FUNCTION_BLOCK FB_teknicMotorEC
VAR
	//I/O
	bBrake			AT %Q*  : BOOL;
	bHomeSensor		AT %I*  : BOOL;
	bClampSensor 	AT %I*  : BOOL;
	fHeightDisp				: REAL;
	
	//Init
	bMotorInverted : BOOL;
	bMotorDisables : BOOL;
	
	fMoveAccl 		: LREAL := 50;
	fMoveDcl 		: LREAL := 50;
	fMoveVelocity 	: LREAL;
	
	torqueVelocity		: LREAL;
	torqueAcceleration	: LREAL;
	torqueDeceleration	: LREAL;
	
	homeVelocity		: LREAL;
	homeSetPosition		: LREAL;
	homeTorqueLimit		: LREAL;
	
	jogTorque			: LREAL;
	
	//State Var
	nMoveState 				: INT;
	nMoveStateTorque		: INT;
	nHomeState				: INT;
	nInitState 				: INT;
	nResetState 			: INT;
	estopState 				: INT := 0; // 0 = Idle, 3 = GearOut, 2 = Stop, 1 = Done
	stopState				: INT;
	
	bIdle 					: BOOL;
	bIdleEnabled 			: BOOL;
	bIdleDisabled 			: BOOL;
	
	fMinHeight				: REAL;
	fMaxHeight 				: REAL := 115;
	fPrevHeight				: REAL;
	bSensorWarning			: BOOL;
	fHeight					: REAL;
	nMoveUpCount			: INT;
	nMoveDownCount			: INT;

	stError : ST_errorRef;
	
	// Timer to turn brake on if motor is left holding carriage for so long;
	fbBrakeTimer 	: TON;
	bIn				: BOOL;
	tPt				: TIME := T#1M;
	bQ				: BOOL;
	tEt				: TIME;
	
	/////////// EC Motor //////////////////////////////////
	fbMotor : axis_REF;
	
	//Power
	fbMotorPower	: MC_Power;
	stMotorPowerOut : ST_McOutputs;
	
	//Reset
	fbMotorReset 	: MC_RESET;
	stMotorResetOut : ST_McOutputs;

	//Halt
	fbMotorHalt 	: MC_HALT;
	stMotorHaltOut 	: ST_McOutputs;
	
	//Velocity Jog
	fbMotorJog 		: MC_JOG;
	stMotorJogOut 	: ST_McOutputs;
	eJogMode 		: E_JogMode;
	nJogModeSelect 	: INT := 2;
	

	//Homing
	fbMotorHome		: MC_Home;
	stHomingOptions : ST_HomingOptions;
	stMotorHomeOut 	: ST_McOutputs;
	bDummyHomingCam : BOOL;
	stHomingMode 	: MC_HomingMode;
	bCheckhomeSensor: BOOL;
	bMotorHomeStatus: BOOL;
	bHomeSensorTriggered : BOOL;
	fbFreeSensorTimer : TON;
	
	//Mode
	fbMotorWriteMode	: MC_WriteDriveOperationMode;
	stMotorWriteModeOut : ST_McOutputs;
	fbMotorReadMode		: MC_ReadDriveOperationMode;
	stMotorReadModeOut 	: ST_McOutputs;
	stOpModeMotor 		: E_DriveOperationMode;
	stOpModeMotorInt	: DINT;
	stWriteMode 		: E_DriveOperationMode;
	nWriteModeSelect 	: DINT := 0;
	fbReadBoolParam		: MC_readParameter;
	fbReadRealParam		: MC_readParameter;
	stReadParamOut 		: ST_mcOutputs;
	eParameter 			: MC_AxisParameter; //Parameter to read or write. https://infosys.beckhoff.com/english.php?content=../content/1033/tcplclib_tc2_mc2/70069259.html&id=
	fReadValue 			: LREAL; // Return value when MC_AxisParameter is of type REAL
	bReadValue 			: LREAL; // Return value when MC_AxisParameter is of type BOOL
	fbWriteRealParam	: MC_WriteParameter;
	fbWriteBoolParam	: MC_WriteParameter;
	stWriteParameterOut : ST_mcOutputs;
	fWriteValue 		: LREAL; // Write value when MC_AxisParameter is of type REAL
	bWriteValue			: BOOL; // Write value when MC_AxisParameter is of type BOOL
	
	//Move Absolute
	fbMotorMoveAbsolute		: MC_MoveAbsolute;
	stMotorMoveAbsoluteOut 	: ST_mcOutputs;
	bChangePosition 		: BOOL;
	fPosition 				: LREAL := 300;
	fStartPos				: LREAL;
	fHalfwayPos				: LREAL;
	
	//Move Relative
	fbMotorMoveRelative		: MC_MoveRelative;
	stMotorMoveRelativeOut 	: ST_McOutputs;
	
	//Move Velocity
	fbMotorMoveVelocity		: MC_MoveVelocity;
	stMotorMoveVelocityOut	: ST_mcOutputs;
	fVel 					: LREAL := 100;
	stDirection 			: MC_Direction;
	stDirectionSelect 		: INT := 1;

	// Stop
	fbMotorStop		: MC_Stop;
	stMotorStopOut 	: ST_mcOutputs;
	bExectuteStop 	: BOOL;
	bStopDone 		: BOOL;
	bStopBtn 		: BOOL;
	
	//Torque
	fbMotorTorque		: FB_moveToTorque;
	stMotorTorqueOut 	: ST_mcOutputs;
	fTorque 			: LREAL := 2;
	torqueDirection		: INT;
	torqueTime			: TIME := T#200MS;

	
	//Gear Coupling
	fbMotorGearIn : MC_GearIn;
	fbMotorGearOut: MC_GearOut;
	stMotorGearInOut : ST_McOutputs;
	stMotorGearOutOut: ST_McOutputs;
	refMasterAxis : axis_REF;
	
	//Status
	fbMotorReadStatus 		: MC_ReadStatus;
	stMotorStatus 			: ST_AxisStatus;
	stMotorReadStatusOut 	: ST_mcOutputs;
	
	//Set Position
	fbMotorSetPosition			: MC_SetPosition;
	stMotorSetPositionOut 		: ST_mcOutputs;
	stMotorSetPositionOption 	: ST_SetPositionOptions;

	fbMotorWriteParameter	: MC_WriteParameter;
	stMotorWriteOut 		: ST_mcOutputs;
	
	sModeDisp 		: STRING;
	fbReadModeTimer	: TON;
		
	fbHomeToTorque		: FB_homeToTorque;
	stHomeToTorqueOut 	: ST_mcOutputs;
	direction			: INT; // 0- PositiveDirection, 1- NegativeDirection
	homeTimeLimit		: TIME := T#2M;
	//homeBackOffPos		: LREAL := 1.5;
	homeBackOffPos		: LREAL := 10;

	bUsingStopReset: BOOL;
END_VAR

(* Behavior of this motor setup is a steady state of disabling the motor when no command is being executed. This setup is best with motors that have a brake
connected to the PLC or motors connected to systems where the system can remain still without assistance from the motor. 
*)
fbBrakeTimer(IN:= bIn, PT:= tPt, Q=> bQ, ET=> tEt);
IF GVL_machine.bMotorsInitialized AND nResetState = 0 THEN
	//bUsingStopReset := FALSE;
	IF bIdleDisabled THEN 
		bIn := TRUE;
	ELSE
		bIn := FALSE;
	END_IF
	
	IF bQ THEN
		IF fbMotor.status.HasJob THEN 
			bIn := FALSE;
		ELSE
			stop();
			brakeOn();
		END_IF
		
	END_IF
	
	(*IF bIdle THEN
		bIdleDisabled R= bIdle;
		bIdleEnabled S= SEL(stop() = 1,FALSE,TRUE);
	ELSE
		bIdleEnabled R= NOT bIdle;
		bIdleDisabled S= SEL(removeStop() = 1,FALSE,TRUE);
	END_IF*)
	IF bIdle THEN
		bIdleDisabled R= bIdle;
		IF (fbMotor.Status.HasBeenStopped OR fbMotor.Status.StandStill) AND bIdleEnabled THEN
			stopState := 0;
			fbMotorStop.Execute := FALSE;
		ELSE
			bIdleEnabled := SEL(stop() = 1,FALSE,TRUE);
			//bUsingStopReset := TRUE;
		END_IF
	ELSE
		bIdleEnabled R= NOT bIdle;
		IF (fbMotor.Status.HasBeenStopped OR fbMotor.Status.StandStill) AND NOT bIdleDisabled THEN
			bIdleDisabled := SEL(removeStop() = 1,FALSE,TRUE);
		ELSE
			stopState := 0;
		END_IF
	END_IF
END_IF

	
actPower();
actHome();
actMode();
actStop();
actMove();
actTorque();
actCouple();
actStatus();


fbMotor();
fbMotorJog.JogForward := FALSE;
fbMotorJog.JogBackwards := FALSE;

ACTION actCouple:
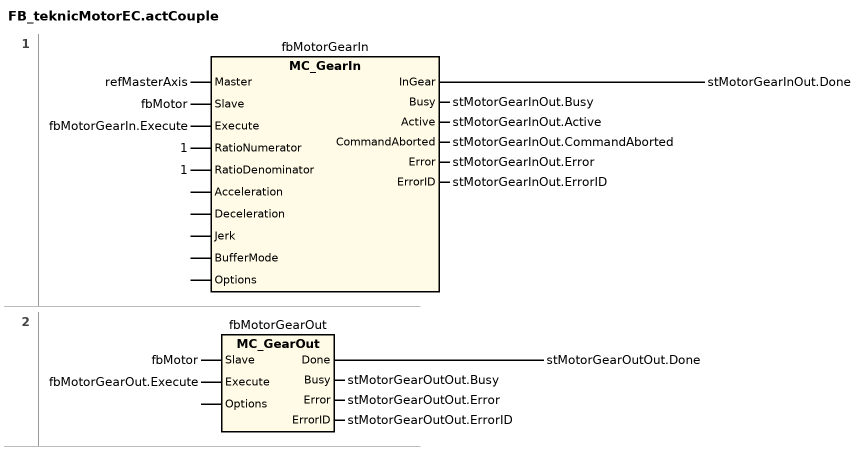
// NETWORK 1
fbMotorGearIn(
    Master := refMasterAxis,
    Slave := fbMotor,
    Execute := fbMotorGearIn.Execute,
    RatioNumerator := 1,
    RatioDenominator := 1,
    Busy => stMotorGearInOut.Busy,
    Active => stMotorGearInOut.Active,
    CommandAborted => stMotorGearInOut.CommandAborted,
    Error => stMotorGearInOut.Error,
    ErrorID => stMotorGearInOut.ErrorID); // MC_GearIn
stMotorGearInOut.Done := fbMotorGearIn.InGear;

// NETWORK 2
fbMotorGearOut(
    Slave := fbMotor,
    Execute := fbMotorGearOut.Execute,
    Busy => stMotorGearOutOut.Busy,
    Error => stMotorGearOutOut.Error,
    ErrorID => stMotorGearOutOut.ErrorID); // MC_GearOut
stMotorGearOutOut.Done := fbMotorGearOut.Done;
END_ACTION

ACTION actHome:
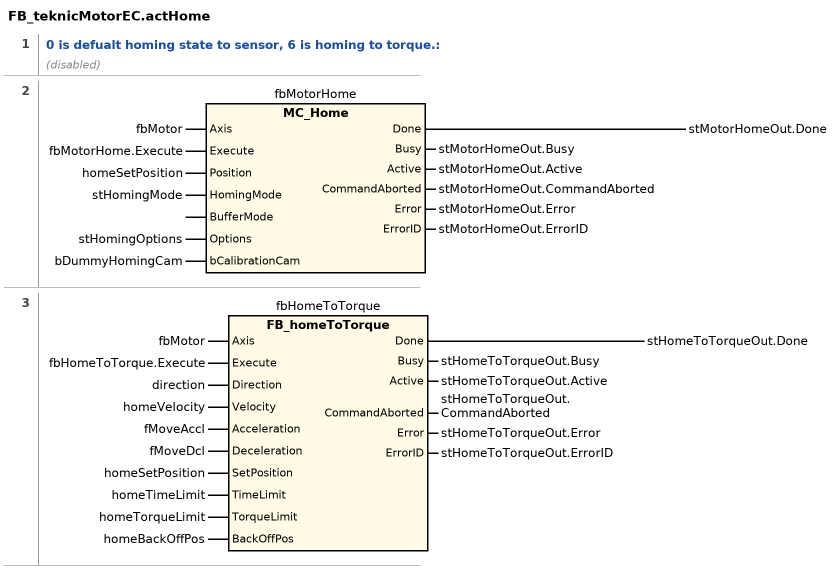
// NETWORK 1 (disabled)
// label: 0 is defualt homing state to sensor, 6 is homing to torque.

// NETWORK 2
fbMotorHome(
    Axis := fbMotor,
    Execute := fbMotorHome.Execute,
    Position := homeSetPosition,
    HomingMode := stHomingMode,
    Options := stHomingOptions,
    bCalibrationCam := bDummyHomingCam,
    Busy => stMotorHomeOut.Busy,
    Active => stMotorHomeOut.Active,
    CommandAborted => stMotorHomeOut.CommandAborted,
    Error => stMotorHomeOut.Error,
    ErrorID => stMotorHomeOut.ErrorID); // MC_Home
stMotorHomeOut.Done := fbMotorHome.Done;

// NETWORK 3
fbHomeToTorque(
    Axis := fbMotor,
    Execute := fbHomeToTorque.Execute,
    Direction := direction,
    Velocity := homeVelocity,
    Acceleration := fMoveAccl,
    Deceleration := fMoveDcl,
    SetPosition := homeSetPosition,
    TimeLimit := homeTimeLimit,
    TorqueLimit := homeTorqueLimit,
    BackOffPos := homeBackOffPos,
    Busy => stHomeToTorqueOut.Busy,
    Active => stHomeToTorqueOut.Active,
    CommandAborted => stHomeToTorqueOut.CommandAborted,
    Error => stHomeToTorqueOut.Error,
    ErrorID => stHomeToTorqueOut.ErrorID); // FB_homeToTorque
stHomeToTorqueOut.Done := fbHomeToTorque.Done;
END_ACTION

ACTION actMode:
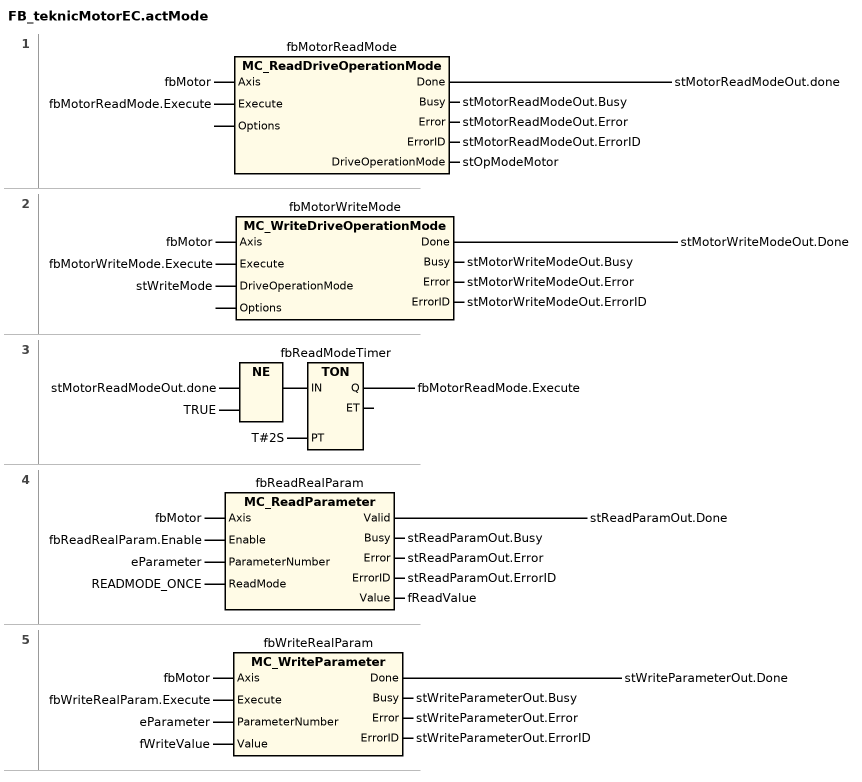
// NETWORK 1
fbMotorReadMode(
    Axis := fbMotor,
    Execute := fbMotorReadMode.Execute,
    Busy => stMotorReadModeOut.Busy,
    Error => stMotorReadModeOut.Error,
    ErrorID => stMotorReadModeOut.ErrorID,
    DriveOperationMode => stOpModeMotor); // MC_ReadDriveOperationMode
stMotorReadModeOut.done := fbMotorReadMode.Done;

// NETWORK 2
fbMotorWriteMode(
    Axis := fbMotor,
    Execute := fbMotorWriteMode.Execute,
    DriveOperationMode := stWriteMode,
    Busy => stMotorWriteModeOut.Busy,
    Error => stMotorWriteModeOut.Error,
    ErrorID => stMotorWriteModeOut.ErrorID); // MC_WriteDriveOperationMode
stMotorWriteModeOut.Done := fbMotorWriteMode.Done;

// NETWORK 3
fbReadModeTimer(IN := stMotorReadModeOut.done <> TRUE, PT := T#2S); // TON
fbMotorReadMode.Execute := fbReadModeTimer.Q;

// NETWORK 4
fbReadRealParam(
    Axis := fbMotor,
    Enable := fbReadRealParam.Enable,
    ParameterNumber := eParameter,
    ReadMode := READMODE_ONCE,
    Busy => stReadParamOut.Busy,
    Error => stReadParamOut.Error,
    ErrorID => stReadParamOut.ErrorID,
    Value => fReadValue); // MC_ReadParameter
stReadParamOut.Done := fbReadRealParam.Valid;

// NETWORK 5
fbWriteRealParam(
    Axis := fbMotor,
    Execute := fbWriteRealParam.Execute,
    ParameterNumber := eParameter,
    Value := fWriteValue,
    Busy => stWriteParameterOut.Busy,
    Error => stWriteParameterOut.Error,
    ErrorID => stWriteParameterOut.ErrorID); // MC_WriteParameter
stWriteParameterOut.Done := fbWriteRealParam.Done;
END_ACTION

ACTION actMove:
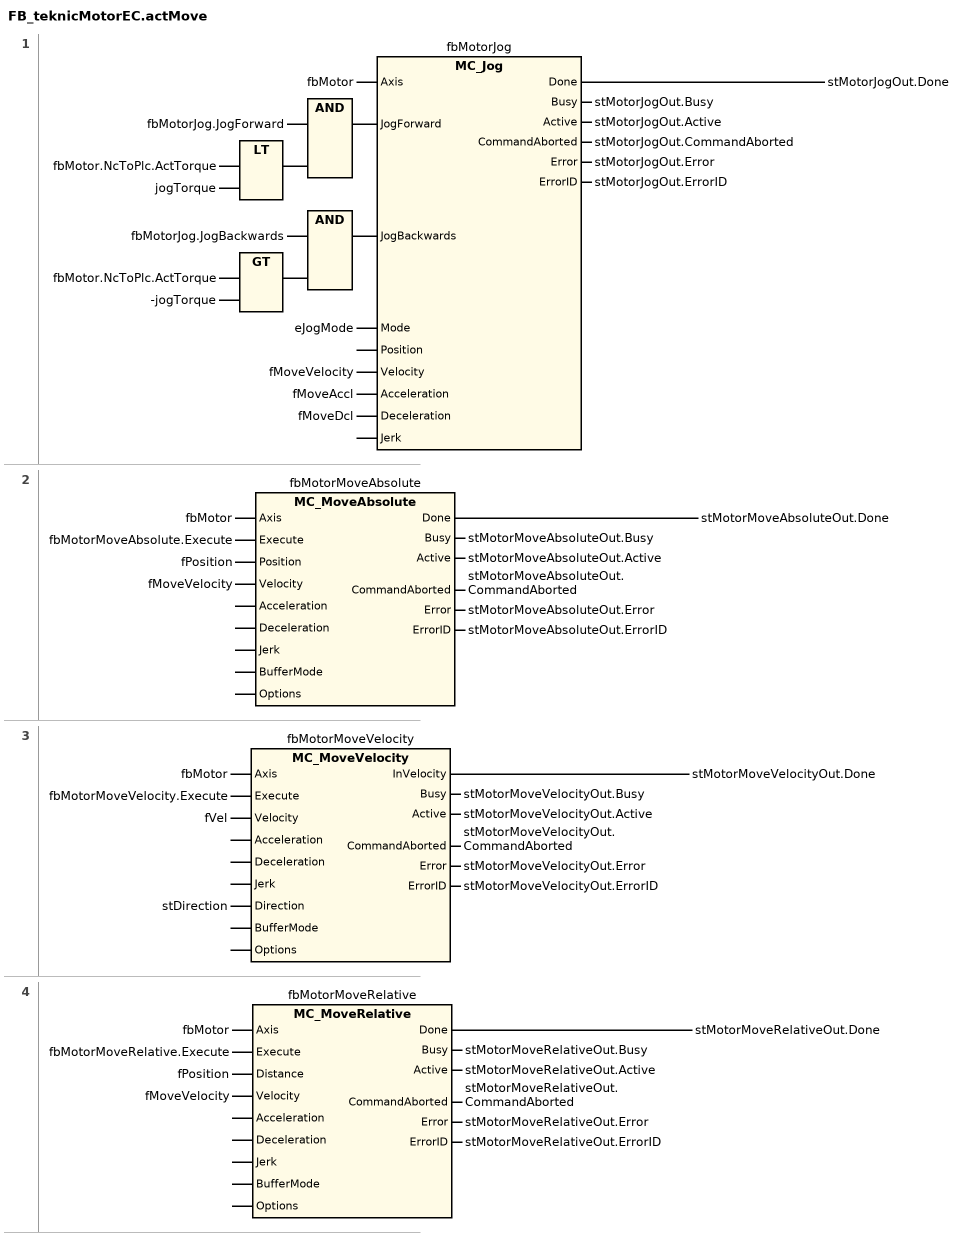
// NETWORK 1
fbMotorJog(
    Axis := fbMotor,
    JogForward := fbMotorJog.JogForward AND fbMotor.NcToPlc.ActTorque < jogTorque,
    JogBackwards := fbMotorJog.JogBackwards AND fbMotor.NcToPlc.ActTorque > (-jogTorque),
    Mode := eJogMode,
    Velocity := fMoveVelocity,
    Acceleration := fMoveAccl,
    Deceleration := fMoveDcl,
    Busy => stMotorJogOut.Busy,
    Active => stMotorJogOut.Active,
    CommandAborted => stMotorJogOut.CommandAborted,
    Error => stMotorJogOut.Error,
    ErrorID => stMotorJogOut.ErrorID); // MC_Jog
stMotorJogOut.Done := fbMotorJog.Done;

// NETWORK 2
fbMotorMoveAbsolute(
    Axis := fbMotor,
    Execute := fbMotorMoveAbsolute.Execute,
    Position := fPosition,
    Velocity := fMoveVelocity,
    Busy => stMotorMoveAbsoluteOut.Busy,
    Active => stMotorMoveAbsoluteOut.Active,
    CommandAborted => stMotorMoveAbsoluteOut.CommandAborted,
    Error => stMotorMoveAbsoluteOut.Error,
    ErrorID => stMotorMoveAbsoluteOut.ErrorID); // MC_MoveAbsolute
stMotorMoveAbsoluteOut.Done := fbMotorMoveAbsolute.Done;

// NETWORK 3
fbMotorMoveVelocity(
    Axis := fbMotor,
    Execute := fbMotorMoveVelocity.Execute,
    Velocity := fVel,
    Direction := stDirection,
    Busy => stMotorMoveVelocityOut.Busy,
    Active => stMotorMoveVelocityOut.Active,
    CommandAborted => stMotorMoveVelocityOut.CommandAborted,
    Error => stMotorMoveVelocityOut.Error,
    ErrorID => stMotorMoveVelocityOut.ErrorID); // MC_MoveVelocity
stMotorMoveVelocityOut.Done := fbMotorMoveVelocity.InVelocity;

// NETWORK 4
fbMotorMoveRelative(
    Axis := fbMotor,
    Execute := fbMotorMoveRelative.Execute,
    Distance := fPosition,
    Velocity := fMoveVelocity,
    Busy => stMotorMoveRelativeOut.Busy,
    Active => stMotorMoveRelativeOut.Active,
    CommandAborted => stMotorMoveRelativeOut.CommandAborted,
    Error => stMotorMoveRelativeOut.Error,
    ErrorID => stMotorMoveRelativeOut.ErrorID); // MC_MoveRelative
stMotorMoveRelativeOut.Done := fbMotorMoveRelative.Done;
END_ACTION

ACTION actPower:
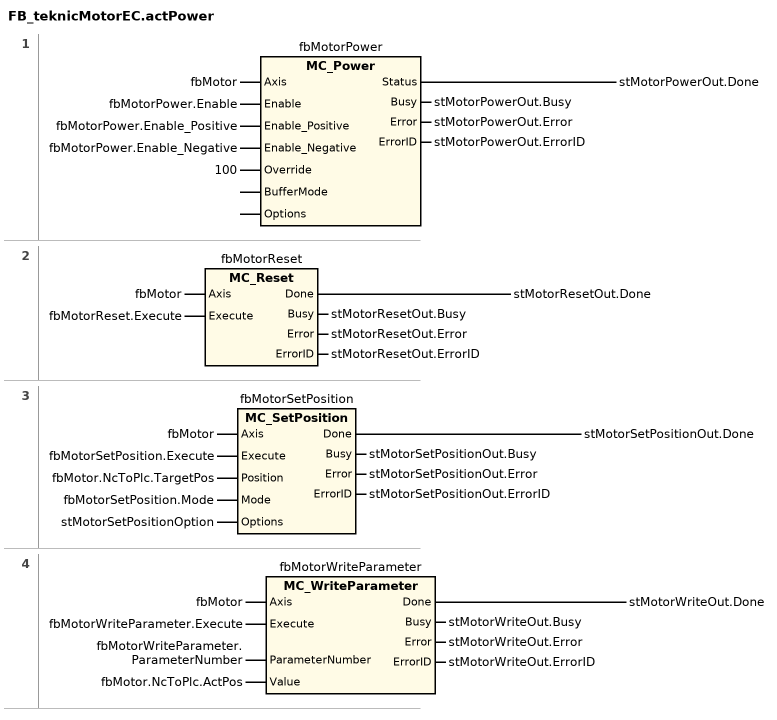
// NETWORK 1
fbMotorPower(
    Axis := fbMotor,
    Enable := fbMotorPower.Enable,
    Enable_Positive := fbMotorPower.Enable_Positive,
    Enable_Negative := fbMotorPower.Enable_Negative,
    Override := 100,
    Busy => stMotorPowerOut.Busy,
    Error => stMotorPowerOut.Error,
    ErrorID => stMotorPowerOut.ErrorID); // MC_Power
stMotorPowerOut.Done := fbMotorPower.Status;

// NETWORK 2
fbMotorReset(
    Axis := fbMotor,
    Execute := fbMotorReset.Execute,
    Busy => stMotorResetOut.Busy,
    Error => stMotorResetOut.Error,
    ErrorID => stMotorResetOut.ErrorID); // MC_Reset
stMotorResetOut.Done := fbMotorReset.Done;

// NETWORK 3
fbMotorSetPosition(
    Axis := fbMotor,
    Execute := fbMotorSetPosition.Execute,
    Position := fbMotor.NcToPlc.TargetPos,
    Mode := fbMotorSetPosition.Mode,
    Options := stMotorSetPositionOption,
    Busy => stMotorSetPositionOut.Busy,
    Error => stMotorSetPositionOut.Error,
    ErrorID => stMotorSetPositionOut.ErrorID); // MC_SetPosition
stMotorSetPositionOut.Done := fbMotorSetPosition.Done;

// NETWORK 4
fbMotorWriteParameter(
    Axis := fbMotor,
    Execute := fbMotorWriteParameter.Execute,
    ParameterNumber := fbMotorWriteParameter.ParameterNumber,
    Value := fbMotor.NcToPlc.ActPos,
    Busy => stMotorWriteOut.Busy,
    Error => stMotorWriteOut.Error,
    ErrorID => stMotorWriteOut.ErrorID); // MC_WriteParameter
stMotorWriteOut.Done := fbMotorWriteParameter.Done;
END_ACTION

ACTION actStatus:
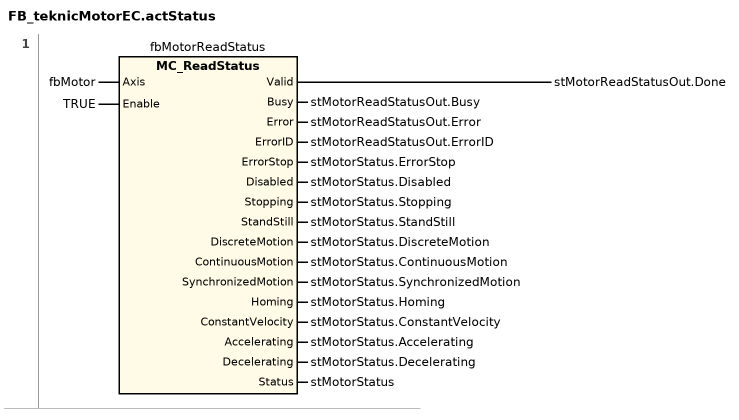
// NETWORK 1
fbMotorReadStatus(
    Axis := fbMotor,
    Enable := TRUE,
    Busy => stMotorReadStatusOut.Busy,
    Error => stMotorReadStatusOut.Error,
    ErrorID => stMotorReadStatusOut.ErrorID,
    ErrorStop => stMotorStatus.ErrorStop,
    Disabled => stMotorStatus.Disabled,
    Stopping => stMotorStatus.Stopping,
    StandStill => stMotorStatus.StandStill,
    DiscreteMotion => stMotorStatus.DiscreteMotion,
    ContinuousMotion => stMotorStatus.ContinuousMotion,
    SynchronizedMotion => stMotorStatus.SynchronizedMotion,
    Homing => stMotorStatus.Homing,
    ConstantVelocity => stMotorStatus.ConstantVelocity,
    Accelerating => stMotorStatus.Accelerating,
    Decelerating => stMotorStatus.Decelerating,
    Status => stMotorStatus); // MC_ReadStatus
stMotorReadStatusOut.Done := fbMotorReadStatus.Valid;
END_ACTION

ACTION actStop:
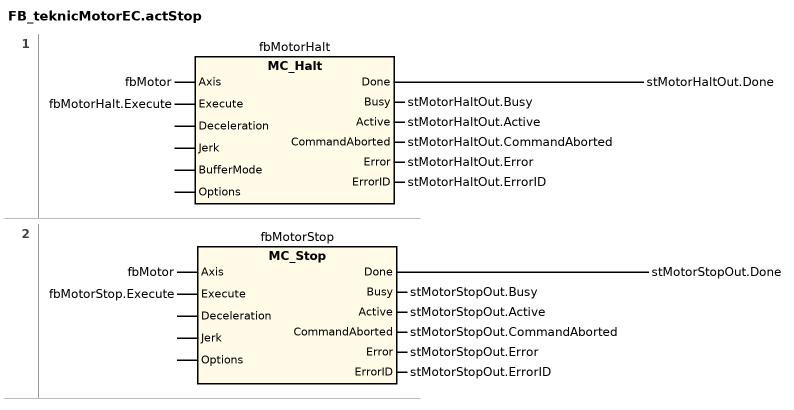
// NETWORK 1
fbMotorHalt(
    Axis := fbMotor,
    Execute := fbMotorHalt.Execute,
    Busy => stMotorHaltOut.Busy,
    Active => stMotorHaltOut.Active,
    CommandAborted => stMotorHaltOut.CommandAborted,
    Error => stMotorHaltOut.Error,
    ErrorID => stMotorHaltOut.ErrorID); // MC_Halt
stMotorHaltOut.Done := fbMotorHalt.Done;

// NETWORK 2
fbMotorStop(
    Axis := fbMotor,
    Execute := fbMotorStop.Execute,
    Busy => stMotorStopOut.Busy,
    Active => stMotorStopOut.Active,
    CommandAborted => stMotorStopOut.CommandAborted,
    Error => stMotorStopOut.Error,
    ErrorID => stMotorStopOut.ErrorID); // MC_Stop
stMotorStopOut.Done := fbMotorStop.Done;
END_ACTION

ACTION actTorque:
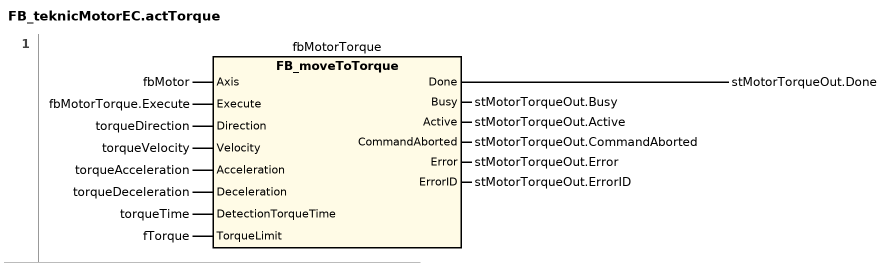
// NETWORK 1
fbMotorTorque(
    Axis := fbMotor,
    Execute := fbMotorTorque.Execute,
    Direction := torqueDirection,
    Velocity := torqueVelocity,
    Acceleration := torqueAcceleration,
    Deceleration := torqueDeceleration,
    DetectionTorqueTime := torqueTime,
    TorqueLimit := fTorque,
    Busy => stMotorTorqueOut.Busy,
    Active => stMotorTorqueOut.Active,
    CommandAborted => stMotorTorqueOut.CommandAborted,
    Error => stMotorTorqueOut.Error,
    ErrorID => stMotorTorqueOut.ErrorID); // FB_moveToTorque
stMotorTorqueOut.Done := fbMotorTorque.Done;
END_ACTION

METHOD brakeOff : BOOL
VAR_INPUT
END_VAR
bBrake := TRUE;
END_METHOD

METHOD brakeOn : BOOL
VAR_INPUT
END_VAR
bBrake := FALSE;
END_METHOD

PROPERTY camSensor : BOOL
GET
camSensor := bDummyHomingCam;
END_GET
END_PROPERTY

METHOD checkOutputs : INT
VAR_INPUT
	stRefFB : REFERENCE TO ST_McOutputs;
END_VAR
checkOutputs := 0;
IF stRefFB.Error THEN
	checkOutputs := 13;
ELSIF stRefFB.Done THEN
	checkOutputs := 1;	
ELSIF stRefFB.Active THEN
	checkOutputs := 2;
ELSIF stRefFB.Busy THEN 
	checkOutputs := 3;
ELSIF stRefFB.CommandAborted THEN
	checkOutputs := 4;
END_IF
END_METHOD

METHOD coupleToAxis : INT
VAR_INPUT
	refMasterAxisIn : REFERENCE TO axis_REF; // Master axis to couple current axis too. 
END_VAR
coupleToAxis := 0;
refMasterAxis := refMasterAxisIn;
bIdle := FALSE;
motorIdle := FALSE;
IF bIdleDisabled THEN
	fbMotorGearIn.Execute := TRUE;
	CASE checkOutputs(stMotorGearInOut) OF 
		1:// Done
			fbMotorGearIn.Execute := FALSE;
			coupleToAxis := 1;
		2:// Active	
		3:// Busy
		4:// Command Aborted
		13:// Error
			stError.errorState := MCGEARIN;
			stError.errorLoc := 'Height Motor coupleToAxis';
			setError(stMotorGearInOut);
			coupleToAxis := 13;
	END_CASE 
ELSE
	fbMotorGearIn.Execute := FALSE;
END_IF
END_METHOD

METHOD decoupleAxis : INT
VAR_INPUT
END_VAR
decoupleAxis := 0;
fbMotorGearIn.Execute := FALSE;
fbMotorGearOut.Execute := TRUE;
CASE checkOutputs(stMotorGearOutOut) OF 
	1:// Done
		fbMotorGearOut.Execute := FALSE;
		decoupleAxis := 1;
	2:// Active	
	3:// Busy
	4:// Command Aborted
	13:// Error
		stError.errorState := MCGEAROUT;
		stError.errorLoc := 'Height Motor decoupleAxis';
		setError(stMotorGearOutOut);
		decoupleAxis := 13;
END_CASE 

stop();
END_METHOD

METHOD disable : INT
VAR_INPUT
END_VAR
disable := 0;
fbMotorPower.Enable := FALSE;
fbMotorPower.Enable_Negative := FALSE;
fbMotorPower.Enable_Positive := FALSE;

IF NOT stMotorPowerOut.Busy AND NOT stMotorPowerOut.Active THEN 
	brakeOn();
	fbMotorPower.Enable := FALSE;
	disable := 1;
ELSIF stMotorPowerOut.Error THEN
	stError.errorState := MCPOWER;
	stError.errorLoc :=  'teknicMotorHeight_disable';
	setError(stMotorPowerOut);
	disable := 13;
END_IF
END_METHOD

PROPERTY distance : REAL;
GET
distance := fbMotor.NcToPlc.ActPos;
END_GET
END_PROPERTY

METHOD enable : INT //1: done, 2: Busy , 13: error
VAR_INPUT
END_VAR
enable := 0;
fbMotorPower.Enable := TRUE;
fbMotorPower.Enable_Negative := TRUE;
fbMotorPower.Enable_Positive := TRUE;

CASE checkOutputs(stMotorPowerOut) OF 
	13:// Error
		enable := 13;
	3:// Busy
		enable := 2;
	1:// Done
		enable := 1;
END_CASE
END_METHOD

METHOD estop : INT
VAR_INPUT
END_VAR
(*
estop := 0;
IF fbMotor.Status.Coupled THEN
	decoupleAxis();
ELSE 
	fbMotorStop.Execute := TRUE;
	
	CASE checkOutputs(stMotorStopOut) OF 
		1:// Done
			brakeOn();
			fbMotorPower.Enable := FALSE;
			estop := 1;
		2:// Active
		3:// Busy
		4:// Command Aborted
		13:// Error
			stError.errorState := MCSTOP;
			stError.errorLoc := 'Height Motor Stop';
			setError(stMotorStopOut);
			estop := 13;
	END_CASE
END_IF
*)
estop := 0;

CASE estopState OF
    0: // Start estop
        IF fbMotor.Status.Coupled THEN
            decoupleAxis();
            estopState := 1;
        ELSE
            fbMotorStop.Execute := TRUE;
            estopState := 2;
        END_IF

    1: // Wait for GearOut.Done
        decoupleAxis();
        IF decoupleAxis() = 1 THEN
            fbMotorStop.Execute := TRUE;
            estopState := 2;
        ELSIF decoupleAxis() = 13 THEN
            estop := 13;
            estopState := 0;
        END_IF

    2: // Wait for MC_Stop.Done
        CASE checkOutputs(stMotorStopOut) OF 
            1: // Done
                brakeOn();
                fbMotorPower.Enable := FALSE;
                estop := 1;
                estopState := 0;
            2: // Active
            3: // Busy
            4: // Command Aborted
            13: // Error
                stError.errorState := MCSTOP;
                stError.errorLoc := 'Height Motor Stop';
                setError(stMotorStopOut);
                estop := 13;
                estopState := 0;
        END_CASE

    3: // Done
        // estop complete — remain here or reset estopState externally
END_CASE
END_METHOD

METHOD homeSetToCount : INT //0:Not done, 1:done, 13: error
VAR_INPUT
	count : LREAL; // Homing that sets count to motor without movement of motor. 
END_VAR
bIdle := FALSE;
IF bIdleDisabled THEN
		//Force motor calibration without move.
		bMotorHomeStatus 	:= TRUE;
		homeSetPosition		:= count;
		stHomingMode 		:= MC_Direct;
		
		fbMotorHome.Execute := TRUE;
		actHome();
		CASE checkOutputs(stMotorHomeOut) OF 
			1:// Done
				fbMotorHome.Execute := FALSE;
				homeSetToCount := 1; 
			2:// Active
				homeSetToCount := 2;
			3:// Busy
			4:// Command Aborted
			13:// Error
				stError.errorState := MCHOME;
				stError.errorLoc := 'homeToZero';
				setError(stMotorHomeOut);
				homeSetToCount := 13;
		END_CASE
	
END_IF
END_METHOD

PROPERTY homeTorqueLimitIn : LREAL
SET
homeTorqueLimit := homeTorqueLimitIn;
END_SET
END_PROPERTY

METHOD homeToSensor : INT //0:Not done, 1:done, 2:Active, 13: error
VAR_INPUT
	stHomingSelect : INT := 0; // 0: Default Homing, 1: Sets the axis position directly to Position without executing a movement --CHANGE fHomingPos to desired Count.
END_VAR

(* Need to figure out torque value for homing.
Need to determine which direction of travel to enable*)
////////////////////////////////////////////////////////////
bIdle := FALSE;
IF bIdleDisabled THEN
	IF NOT bMotorHomeStatus THEN
		fbFreeSensorTimer(PT:=T#1S);
		IF NOT bCheckhomeSensor THEN
 			IF bHomeSensor THEN 
				//Force motor calibration without move.
				bMotorHomeStatus := TRUE;
				stHomingSelect := 2;
				CASE stHomingSelect OF 
					0: stHomingMode := MC_DefaultHoming;
					1: stHomingMode := MC_Direct;
					2: stHomingMode := MC_ForceCalibration;
					3: stHomingMode := MC_ResetCalibration;
				END_CASE
				fbMotorHome.Execute := TRUE;
				actHome();
				CASE checkOutputs(stMotorHomeOut) OF 
					1:// Done
						fbMotorHome.Execute := FALSE;
						homeToSensor := 1; 
					2:// Active
						homeToSensor := 2;
					3:// Busy
					4:// Command Aborted
					13:// Error
						stError.errorState := MCHOME;
						stError.errorLoc := 'homeToSensor_actual';
						setError(stMotorHomeOut);
						homeToSensor := 13;
				END_CASE
			END_IF
			bCheckHomeSensor := TRUE;
		ELSE
			homeToSensor := 0;
			//Homing Mode 
			CASE stHomingSelect OF 
				0: stHomingMode := MC_DefaultHoming;
				1: stHomingMode := MC_Direct;
				2: stHomingMode := MC_ForceCalibration;
				3: stHomingMode := MC_ResetCalibration;
			END_CASE
			fbMotorHome.Execute := TRUE;
			CASE checkOutputs(stMotorHomeOut) OF 
				1:// Done
					fbMotorHome.Execute := FALSE;
					homeToSensor := 1; 
				2:// Active
					homeToSensor := 2;
				3:// Busy
				4:// Command Aborted
				13:// Error
					stError.errorState := MCHOME;
					stError.errorLoc := 'homeToSensor_actual';
					setError(stMotorHomeOut);
					homeToSensor := 13;
			END_CASE
					
			//Homing Sensor trigger (torque)
			IF fbMotorHome.Execute AND NOT bHomeSensorTriggered THEN
				bDummyHomingCam := bHomeSensor;
				IF bHomeSensor THEN
					bHomeSensorTriggered := TRUE;
				END_IF
				
			ELSE
				IF stHomingOptions.SearchDirection = MC_Negative_Direction THEN
					fbFreeSensorTimer.IN := TRUE;
					IF fbFreeSensorTimer.Q THEN
						bDummyHomingCam := FALSE;
					END_IF
				ELSE
					bDummyHomingCam := bHomeSensor;
				END_IF
			END_IF
			
			bMotorHomeStatus := fbMotor.Status.Homed;
		END_IF
	ELSE
		fPosition := 0;
		fbMotorMoveAbsolute.Execute := TRUE;
		CASE checkOutputs(stMotorMoveAbsoluteOut) OF 
			1:// Done
				fbMotorMoveAbsolute.Execute := FALSE;
				bHomeSensorTriggered := FALSE;
				fbFreeSensorTimer(IN := FALSE);
				homeToSensor := 1;
			2:// Active
				homeToSensor := 2;
			3:// Busy
			4:// Command Aborted
				fbMotorMoveAbsolute.Execute := FALSE;
			13:// Error
				stError.errorState := MCMOVEABSOLUTE;
				stError.errorLoc := 'homeToSensor_0';
				setError(stMotorMoveAbsoluteOut);
				homeToSensor := 13;
				fbMotorMoveAbsolute.Execute := FALSE;
		END_CASE
	END_IF
END_IF
END_METHOD

METHOD homeToTorque : INT //0:Not done, 1:done, 2:Active, 13: error
VAR_INPUT
END_VAR

(* Need to figure out torque value for homing.
Need to determine which direction of travel to enable*)
////////////////////////////////////////////////////////////
bIdle := FALSE;
IF bIdleDisabled THEN
	IF NOT bMotorHomeStatus THEN
		homeToTorque := 0;
		
		IF bMotorInverted THEN
			direction := 0;
		ELSE 
			direction := 1;
		END_IF
		
		fbHomeToTorque.Execute := TRUE;
		CASE checkOutputs(stHomeToTorqueOut) OF 
			1:// Done
				fbHomeToTorque.Execute := FALSE;
				bMotorHomeStatus := fbMotor.Status.Homed;
				homeToTorque := 1; 
			2:// Active
				homeToTorque := 2;
			3:// Busy
				homeToTorque := 3;
			4:// Command Aborted
			13:// Error
				stError.errorState := MCHOME;
				stError.errorLoc := 'homeToTorque';
				setError(stHomeToTorqueOut);
				homeToTorque := 13;
		END_CASE
	ELSE
		CASE nHomeState OF 
			0: // Read soft limit switch to set home pos. 
				IF bMotorInverted THEN
					eParameter := AxisMaxSoftPosLimit;
				ELSE 
					eParameter := AxisMinSoftPosLimit;
				END_IF
				
				fbReadRealParam.Enable := TRUE;
				
				IF NOT stReadParamOut.Busy AND stReadParamOut.Done THEN
					fbReadRealParam.Enable := FALSE;
					fPosition := fReadValue;
					nHomeState := nHomeState + 1;
				ELSIF NOT stReadParamOut.Busy AND stReadParamOut.Error THEN
					homeToTorque := 13;
					fbReadRealParam.Enable := FALSE;
					nHomeState := 0;
				END_IF
		
			1: // Execute Move to Home Pos. 
			
			fbMotorMoveAbsolute.Execute := TRUE;
			CASE checkOutputs(stMotorMoveAbsoluteOut) OF 
				1:// Done
					fbMotorMoveAbsolute.Execute := FALSE;
					nHomeState := 0;
					homeToTorque := 1;
				2:// Active
					homeToTorque := 2;
				3:// Busy
					homeToTorque := 3;
				4:// Command Aborted
					fbMotorMoveAbsolute.Execute := FALSE;
					nHomeState := 0;
				13:// Error
					stError.errorState := MCMOVEABSOLUTE;
					stError.errorLoc := 'homeToTorque_0';
					setError(stMotorMoveAbsoluteOut);
					nHomeState := 0;
					homeToTorque := 13;
			END_CASE
		END_CASE
	END_IF
END_IF
END_METHOD

METHOD init : BOOL
VAR_INPUT
	bMotorInvertedIn : BOOL; //True if movement away from home position increases counts negatively
	bMotorDisablesIn : BOOL; //True if motor has a brake attached or does not to be enabled when not moving. 
	
	fMoveAcclIn 		: LREAL;
	fMoveDclIn 			: LREAL;
	fMoveVelocityIn 	: LREAL;
	
	torqueVelocityIn		: LREAL;
	torqueAccelerationIn	: LREAL;
	torqueDecelerationIn	: LREAL;
	
	homeVelocityIn			: LREAL; //Homing velocity when homing when using homeToTorque method.
	homeSetPositionIn		: LREAL; //Counts to set encoder when any homing method is complete. 
	homeTorqueLimitIn		: LREAL; //Torque limit to home to when using homeToTorque method. 
	
	jogTorqueIn				: LREAL; // Torque used to limit jog moves. 
END_VAR
init := FALSE;
CASE nInitState OF 
	0: //Reset all function blocks 
		IF resetMotorCommands() THEN
			fbMotorPower.Enable := FALSE;
			nInitState := 5;
		END_IF
	5: // Enable Motor
		CASE enable() OF 
			1:// Done
				nInitState := 6;
			2:// Busy	
			13:// Error
				SetError(stMotorPowerOut);
				stError.errorState := MCPOWER;
				nInitState := 10;
		END_CASE
	6: //Set Init Vars
		bMotorInverted := bMotorInvertedIn;
		bMotorDisables := bMotorDisablesIn;
		
		fMoveAccl 		:= fMoveAcclIn;
		fMoveDcl 		:= fMoveDclIn;
		fMoveVelocity 	:= fMoveVelocityIn;
    	
		torqueVelocity		:= torqueVelocityIn;
		torqueAcceleration	:= torqueAccelerationIn;
		torqueDeceleration	:= torqueDecelerationIn;
		
		homeVelocity		:= homeVelocityIn;
		
		homeSetPosition		:= homeSetPositionIn;
		homeTorqueLimit		:= homeTorqueLimitIn;
		
		jogTorque := jogTorqueIn;
		
		IF NOT bMotorInverted THEN
			stHomingOptions.SearchDirection := MC_Negative_Direction;
		END_IF
		
		nInitState := 0;
		init := TRUE;
		
	7:// Write homing velocity
	
	
	10:// Error			
		CASE reset() OF 
			1:// Done
				nInitState := 0;
			13:// Error
				nInitState := 0;
		END_CASE
END_CASE
END_METHOD

PROPERTY isBusy : BOOL
GET
isBusy := fbMotor.Status.HasJob;
END_GET
END_PROPERTY

PROPERTY isEnabled : BOOL
GET
isEnabled := NOT fbMotor.Status.Disabled;
END_GET
END_PROPERTY

PROPERTY isMotorInverted : BOOL
GET
isMotorInverted := bMotorInverted;
END_GET
END_PROPERTY

PROPERTY isStopped : BOOL
GET
isStopped := fbMotor.Status.HasBeenStopped;
END_GET
END_PROPERTY

PROPERTY stMotorError : ST_errorRef
GET
motorError.errorId := stError.errorId;
motorError.errorLoc := stError.errorLoc;
motorerror.errorMsg := stError.errorMsg;
motorError.errorState := stError.errorState;
END_GET
END_PROPERTY

PROPERTY motorErrorId : UDINT
GET
motorErrorId := stError.errorId;
END_GET
END_PROPERTY

PROPERTY motorIdle : BOOL
SET
bIdle := motorIdle;
END_SET
END_PROPERTY

METHOD moveTo : INT //0: move not done, 1: Move done, 13: error, 15: move is halway complete
VAR_INPUT
	sState 		: STRING; // *OPTIONAL. Can be used to set the state of the move function (0 is reset, 'NULL' is do nothing);
	fHeightInput : REAL;
END_VAR
//////////////////////////////////////////////////////////////////

IF sState = 'NULL' THEN 
	//Do nothing
ELSE
	nMoveState := STRING_TO_INT(sState);
END_IF
moveTo := 0;
fHeightInput := fHeightInput * 25.4; //Convert inches to mm. 
IF bMotorInverted THEN
	fHeightInput := -fHeightInput;
END_IF

bIdle := FALSE;
IF bIdleDisabled THEN
	CASE nMoveState OF 
		0:// Get Average height of sensor 
			fPosition := fHeightInput;
			fStartPos := fbMotor.NcToPlc.ActPos;
			fHalfwayPos := fStartPos + ((fPosition-fStartPos)*0.75);
			nMoveState := 1;
		
		1:// Execute Move
			fPosition := fHeightInput;
			fbMotorMoveAbsolute.Execute := TRUE;
			CASE checkOutputs(stMotorMoveAbsoluteOut) OF 
				1:// Done
					IF fbMotor.NcToPlc.ActPos < fHeightInput + 1 OR fbMotor.NcToPlc.ActPos > fHeightInput - 1 THEN
						fbMotorMoveAbsolute.Execute := FALSE;
						nMoveState := 0;
						moveTo := 1;
					END_IF
				2,3:// Active,Busy
					moveTo := 2;
					IF ABS(fbMotor.NcToPlc.ActPos) >= ABS(fHalfwayPos) THEN
						moveTo := 15;
					END_IF 
				4:// Command Aborted
					fbMotorMoveAbsolute.Execute := FALSE;
				13:// Error
					stError.errorState := MCMOVEABSOLUTE;
					stError.errorLoc := 'MoveTo';
					setError(stMotorMoveAbsoluteOut);
					nMoveState := 0;
					moveTo := 13;
			END_CASE
			(*IF ABS(fbMotor.NcToPlc.ActPos) >= ABS(fHalfwayPos) THEN
				moveTo := 15;
			END_IF *)
	END_CASE
END_IF
END_METHOD

METHOD moveToJog : INT
VAR_INPUT
	nDirection		: INT; // 0- Negative Moves, 1- Positive Moves
END_VAR
moveToJog := 0;

bIdle := FALSE;
IF bIdleDisabled THEN
	eJogMode := MC_JOGMODE_CONTINOUS;
	fbMotorJog.JogForward := SEL(nDirection = 1,FALSE,TRUE);
	fbMotorJog.JogBackwards := SEL(nDirection = 1,TRUE,FALSE);
	
	CASE checkOutputs(stMotorJogOut) OF 
		1:// Done
		2,3:// Active or Busy	
			moveToJog := 1;
		4:// Command Aborted
		13:// Error
			stError.errorState := MCJOG;
			stError.errorLoc := 'MoveToJog';
			setError(stMotorJogOut);
			moveToJog := 13;
	END_CASE 
END_IF
END_METHOD

METHOD moveToSensor : INT
VAR_INPUT
	nDirection		: INT; // 0- Negative Moves, 1- Positive Moves
END_VAR
moveToSensor := 0;

bIdle := FALSE;
IF bIdleDisabled THEN
	eJogMode := MC_JOGMODE_CONTINOUS;
	fbMotorJog.JogForward := SEL(nDirection = 1,FALSE,TRUE);
	fbMotorJog.JogBackwards := SEL(nDirection = 1,TRUE,FALSE);
	CASE checkOutputs(stMotorJogOut) OF 
		1:// Done
		2,3:// Active or Busy
			IF bClampSensor THEN
				fbMotorJog.JogForward := FALSE;
				fbMotorJog.JogBackwards := FALSE;
				moveToSensor := 1;
			END_IF
		4:// Command Aborted
		13:// Error
			stError.errorState := MCJOG;
			stError.errorLoc := 'MoveToSensor';
			setError(stMotorJogOut);
			moveToSensor := 13;
	END_CASE 
END_IF
END_METHOD

METHOD moveToTorque : INT
VAR_INPUT
	sState 			: STRING; // *OPTIONAL. Can be used to set the state of the move function (0 is reset, 'NULL' is do nothing);
	fTorqueInput 	: REAL; // Percentage of torque to move to.
	nDirection		: INT; //// 0- PositiveDirection, 1- NegativeDirection
END_VAR
IF sState = 'NULL' THEN 
	//Do nothing
ELSE
	nMoveStateTorque := STRING_TO_INT(sState);
END_IF
moveToTorque := 0;
torqueDirection := nDirection;

bIdle := FALSE;
IF bIdleDisabled THEN
	CASE nMoveStateTorque OF 
		0:// Set Torque 
			fTorque := fTorqueInput;
			fbMotorTorque.Execute := FALSE;
			nMoveStateTorque := 1;
			
		1:// Execute Move
			fbMotorTorque.Execute := TRUE;
			CASE checkOutputs(stMotorTorqueOut) OF 
				1:// Done
					fbMotorTorque.Execute := FALSE;
					nMoveStateTorque := 0;
					moveToTorque := 1;
				2:// Active
					moveToTorque := 2;
				3:// Busy
				4:// Command Aborted
					fbMotorTorque.Execute := FALSE;
				13:// Error
					stError.errorState := MCTORQUECONTROL;
					stError.errorLoc := 'MoveToTorque';
					setError(stMotorTorqueOut);
					nMoveStateTorque := 0;
					moveToTorque := 13;
			END_CASE
	END_CASE
END_IF
END_METHOD

METHOD readRealParameter : INT
VAR_INPUT
	parameterIn : MC_AxisParameter; 
END_VAR
readRealParameter := 0;
eParameter := parameterIn;
fbReadRealParam.Enable := TRUE;

CASE checkOutputs(stReadParamOut) OF 	
	1:// Done
		readRealParameter := 1;
	3:// Busy 
		readRealParameter := 2;
	13:// Error
		readRealParameter := 13;	
END_CASE
END_METHOD

METHOD removeStop : INT
VAR_INPUT
END_VAR
removeStop := 0;
IF bMotorDisables THEN
	CASE enable() OF 
		1: // Done
			fbMotorStop.Execute := FALSE;
			IF NOT stMotorStopOut.Busy AND NOT stMotorStopOut.Active THEN 
				brakeOff();
				fbMotorStop.Execute := FALSE;
				removeStop := 1;
			ELSIF stMotorHaltOut.Error THEN
				stError.errorState := MCSTOP;
				stError.errorLoc :=  'teknicMotorHeight_removeStop';
				setError(stMotorStopOut);
				removeStop := 13;
			END_IF
		2: //Busy
		13: //Error
			stError.errorState := MCPOWER;
			stError.errorLoc :=  'teknicMotorHeight_removeStop';
			setError(stMotorPowerOut);
			removeStop := 13;
	END_CASE
ELSE
	fbMotorStop.Execute := FALSE;
IF NOT fbMotor.Status.MotionCommandsLocked THEN
	removeStop := 1;
END_IF

CASE checkOutputs(stMotorPowerOut) OF 
	13:// Error
		removeStop := 13;
END_CASE
END_IF
END_METHOD

METHOD reset : INT //0: reset not done, 1: reset done, 2: Busy, 13: error 
VAR_INPUT
END_VAR
reset := 0;
CASE nResetState OF 
	0: // Remove executes on all motor commands
		resetMotorCommands();
		//bMotorHomeStatus := FALSE;
		nResetState := 3;
	3:// Uncouple Motor
		IF fbMotor.Status.Coupled THEN
			nResetState := 4;
		ELSE
			nResetState := 5;
		END_IF
	4:// Decouple Motor
		CASE decoupleAxis() OF 
			1: // Done
				nResetState := 5;
			13: //Error
				nResetState := 0;
				reset := 13;
		END_CASE
	5://Reset Motor
		fbMotorReset.Execute := TRUE;
		CASE checkOutputs(stMotorResetOut) OF 
			1:// Done
				nResetState := 10;
				fbMotorReset.Execute := FALSE;
			2://Active 
				reset := 2;
			3:// Busy
				reset := 2;
			13:// Error
				setError(stMotorResetOut);
				stError.errorState := MCRESET;
				nResetState := 0;
				reset := 13;
		END_CASE
		
	10: //Motor Off 
		IF stMotorPowerOut.Done OR stMotorPowerOut.Error THEN
			fbMotorPower.Enable := FALSE;
			nResetState := 15;
		ELSE
			nResetState := 15;
		END_IF
		
	15://Power Motor On
		fbMotorPower.Enable := TRUE;
		CASE checkOutputs(stMotorPowerOut) OF
			1: //Done
				nResetState := 0;
				reset := 1;
			13: nResetState := 0;
		END_CASE
	
END_CASE
END_METHOD

METHOD resetMotorCommands : BOOL
VAR_INPUT
END_VAR
resetMotorCommands				:= FALSE;
fbMotorReset.Execute 			:= FALSE;
fbMotorHome.Execute 			:= FALSE;
fbMotorReadMode.Execute  		:= FALSE;
fbMotorWriteMode.Execute 		:= FALSE;
fbMotorHalt.Execute      		:= FALSE;
fbMotorStop.Execute      		:= FALSE;
fbMotorMoveAbsolute.Execute 	:= FALSE;
fbMotorMoveVelocity.Execute 	:= FALSE;
fbMotorMoveRelative.Execute 	:= FALSE;
fbMotorTorque.Execute			:= FALSE;
fbMotorGearIn.Execute			:= FALSE;
fbMotorGearOut.Execute			:= FALSE;
fbMotorJog.JogForward 			:= FALSE;
fbMotorJog.JogBackwards 		:= FALSE;
fbHomeToTorque.Execute			:= FALSE;
fbReadRealParam.Enable 			:= FALSE;
fbWriteRealParam.Execute		:= FALSE;

//Reset FB states
nMoveState 		 := 0;
nMoveStateTorque := 0;
nHomeState		 := 0;
nInitState 		 := 0;
estopState		 := 0;
stopState		 := 0;
resetMotorCommands				:= TRUE;
END_METHOD

METHOD setError : BOOL
VAR_INPUT
	stOutput : REFERENCE TO ST_MCOUTPUTS;
END_VAR
stError.errorId := stOutput.ErrorID;
brakeOn();
END_METHOD

METHOD stop : INT //0: stop not done, 1: stop done; 13: error
VAR_INPUT
END_VAR
(*stop := 0;
fbMotorJog.JogForward 	:= FALSE;
fbMotorJog.JogBackwards := FALSE;
IF stMotorPowerOut.Done THEN
	fbMotorStop.Execute := TRUE;
	fbMotorGearOut.Execute := TRUE;
	CASE checkOutputs(stMotorStopOut) OF 
		1:// Done
			fbMotorGearOut.Execute := FALSE;
			IF bMotorDisables THEN
				brakeOn();
				fbMotorPower.Enable := FALSE;
			END_IF
			stop := 1;
		2:// Active
		3:// Busy
		4:// Command Aborted
		13:// Error
			stError.errorState := MCSTOP;
			stError.errorLoc := 'Height Motor Stop';
			setError(stMotorStopOut);
			stop := 13;
	END_CASE
ELSE
	fbMotorStop.Execute := FALSE;
	stop := 1;
END_IF
*)
stop := 0;
fbMotorJog.JogForward  := FALSE;
fbMotorJog.JogBackwards := FALSE;

CASE stopState OF
    0: // Wait for motor power confirmation
        IF stMotorPowerOut.Done THEN
            fbMotorGearOut.Execute := FALSE;
			fbMotorGearIn.Execute := FALSE;
            stopState := 1;
        ELSE
            stop := 1;
        END_IF

    1: // Wait for GearOut
		fbMotorGearOut.Execute := TRUE;
        IF fbMotorGearOut.Done THEN
            fbMotorGearOut.Execute := FALSE;
            fbMotorStop.Execute := FALSE;
            stopState := 2;
        END_IF

    2: // Wait for Stop
		fbMotorStop.Execute := TRUE;
        CASE checkOutputs(stMotorStopOut) OF 
            1: // Done
                fbMotorStop.Execute := FALSE;
				IF bMotorDisables THEN
            		brakeOn();
                	fbMotorPower.Enable := FALSE;
            	END_IF
				stop := 1;
            	stopState := 0;

            13: // Error
                stError.errorState := MCSTOP;
                stError.errorLoc := 'Height Motor Stop';
                setError(stMotorStopOut);
                stop := 13;
                stopState := 0;
        END_CASE

END_CASE
END_METHOD

METHOD writeRealParameter : INT
VAR_INPUT
	parameterIn : MC_AxisParameter;
	valueIn : LREAL;
END_VAR
writeRealParameter := 0;
eParameter := parameterIn;
fWriteValue := valueIn;
fbWriteRealParam.Execute := TRUE;

CASE checkOutputs(stWriteParameterOut) OF 	
	1:// Done
		writeRealParameter := 1;
	3:// Busy 
		writeRealParameter := 2;
	13:// Error
		writeRealParameter := 13;	
END_CASE
END_METHOD

END_FUNCTION_BLOCK

(* stored: Version 1.1.0.1, ProductVersion 3.1.4024.13
   POU FB_teknicMotorEC: Id {daffd6c9-a64a-45f4-b5fb-4e0db812bcca}, SpecialFunc None
   Action actCouple: Id {a51a389d-e95f-4266-87ae-51dddcc8c39d}
   Action actHome: Id {2daf2441-f6a3-4bd9-96dc-419f675c97a1}
   Action actMode: Id {354840e2-2cef-4629-8354-87b057f6201f}
   Action actMove: Id {125eeb7b-a532-4c5f-9542-469e9c3a32de}
   Action actPower: Id {ce4edf73-3c0b-413e-9913-34eca1b7ce92}
   Action actStatus: Id {d912e5ef-f74e-4927-8f03-681aad253cd9}
   Action actStop: Id {2abda9e6-b471-4a96-9a91-103ff17b514c}
   Action actTorque: Id {c61b4ebc-6581-4865-8448-a6d497ca1155}
   Method brakeOff: Id {83c45466-502d-4e2b-bbef-b577292d6467}
   Method brakeOn: Id {8886d7e6-8426-4129-a159-dbeba141bb4b}
   Property camSensor: Id {9270001d-7746-4250-9d93-0a669bef75e3}
   Get Get: Id {2bbfc3bd-cc2a-4911-af04-3cdc4b685ad4}
   Method checkOutputs: Id {8e044763-1449-45c5-829d-ba44c71af699}
   Method coupleToAxis: Id {5b806679-0004-4345-885e-0cc1ff97455d}
   Method decoupleAxis: Id {b0fd01c1-2b44-4299-a809-e3e8d4419caa}
   Method disable: Id {3037b338-345b-4b60-b338-02caaa02ff4f}
   Property distance: Id {67cd1f99-5285-4dad-addb-ef9df61598c8}
   Get Get: Id {9686ba88-518f-4e5d-a851-3bc1ddd7c80a}
   Method enable: Id {04e6c41f-d75f-47f8-9b15-186c28a8ae3c}
   Method estop: Id {c852613a-5abc-4ac5-bfbf-c1ca8daa6642}
   Method homeSetToCount: Id {88606f33-d5fc-4771-949e-bf4c8ce47cbd}
   Property homeTorqueLimitIn: Id {267a3c5f-090d-4904-b27d-b5af8ce01237}
   Set Set: Id {82a12e77-36d7-47ac-b67a-8f56374dc0d7}
   Method homeToSensor: Id {dc133354-1b8e-489e-84ec-ada86bf51b30}
   Method homeToTorque: Id {daa049df-85ae-4364-90c0-22ed16b32c82}
   Method init: Id {e84cce5b-1783-47b9-a117-3f5262799d85}
   Property isBusy: Id {eedb2e44-a496-4123-a82d-5e6ee38dfd8b}
   Get Get: Id {44fe18d0-7134-4bba-8b1f-7364af502cc8}
   Property isEnabled: Id {ec38bf94-2076-4e64-b561-3fda010a102a}
   Get Get: Id {b094fdff-b232-4b4f-8274-3b4a979bf08b}
   Property isMotorInverted: Id {411e130f-f2e1-42cd-8ed1-9bfc092a429c}
   Get Get: Id {84a09ab3-0c81-4f5e-a5e6-da743c695fa1}
   Property isStopped: Id {bd07a007-c01b-4b1a-a6a1-b79026bb856c}
   Get Get: Id {da7aa38c-fc44-4bce-b5e0-2d57646abfce}
   Property motorError: Id {babce6bb-50c7-432e-860d-1339e3ec4651}
   Get Get: Id {1ad91577-0865-4615-a96b-734299de12c4}
   Property motorErrorId: Id {ed1a26c0-3c18-439f-a430-18c0edd9d273}
   Get Get: Id {61591a72-497b-4758-ab9c-c6fc517b8a98}
   Property motorIdle: Id {1614d8be-9f89-4ff2-9fcf-5f44304cc0ff}
   Set Set: Id {c2f5be72-4c91-4b15-8dab-57a848e1c8f4}
   Method moveTo: Id {8b5ed6bb-3d03-493c-a564-57cca23526b4}
   Method moveToJog: Id {6212539f-8c46-4153-937e-1efe5d581699}
   Method moveToSensor: Id {6f67982c-11a1-4f60-b154-c4a0910e50d0}
   Method moveToTorque: Id {2150b389-bcb3-4ce4-9f5c-2c7cf1e3b9ff}
   Method readRealParameter: Id {d970bc4e-75bd-440d-8d04-18e312ef8a77}
   Method removeStop: Id {3815df2a-7092-4177-b9b4-ec0a2c7439fe}
   Method reset: Id {fa32862e-6635-4c70-bb73-2e1626398a76}
   Method resetMotorCommands: Id {58d0bedf-900b-411a-9b2f-dd01c3093275}
   Method setError: Id {0324a971-0b2f-4d11-be9a-fd1a0b7d0d4e}
   Method stop: Id {ca1bcbd3-5151-4386-a120-148a35dc2daf}
   Method writeRealParameter: Id {7f8a080a-cb42-492d-b4da-5aba7c8c4e82} *)
